Universal Robots PolyScope program: c_str.urp

Program c_str (installation=ext_control directory=/programs createdIn=5.17.3 lastSavedIn=5.17.3 robotSerialNumber=20245501435)
Calibrated DH parameters: a=[0.000154, -0.137004, -0.385524, -0.00002, 0.000092, 0]; d=[0.162441, 211.794786, -230.585024, 18.923638, 0.099786, 0.09951]; alpha=[1.569493, -0.001902, 0.003874, 1.570111, -1.570167, 0]; deltaTheta=[0, -1.242934, 1.056292, 0.186646, 0.000002, 0.000001]
InitVariablesNode
Robot Program (runOnlyOnce=false)
  MoveL speed 250 mm/s, acceleration 1200 mm/s^2 (useActiveTCP=true) feature=Base
    Waypoint Waypoint_1: TCP in base x=222.973 y=562.956 z=73.09 mm, rx=-1.7404 ry=-1.5254 rz=0.3572 rad; joints [-130.567, -31.955, 101.515, -146.824, -42.301, -128.37] deg; TCP offset x=28.21 y=-96.107 z=-99.69 mm, rx=0 ry=0 rz=0 rad
    Waypoint Waypoint_2 (Relative): relativeFromPosition TCP in base x=225.604 y=562.943 z=77.706 mm, rx=-1.7406 ry=-1.5243 rz=0.3485 rad; joints [-130.763, -32.421, 101.483, -146.672, -42.264, -128.37] deg; TCP in base x=108.241 y=170.343 z=-59.719 mm, rx=-1.3852 ry=-1.4777 rz=0.7367 rad; joints [-170.461, -4.85, 143.353, -161.62, -71.094, -186.243] deg
